// SIMATIC S7-200 project (STEP 7-Micro/WIN), CPU 224XP CN REL 02.01

ORGANIZATION_BLOCK MAIN:OB1
TITLE=PROGRAM COMMENTS
BEGIN
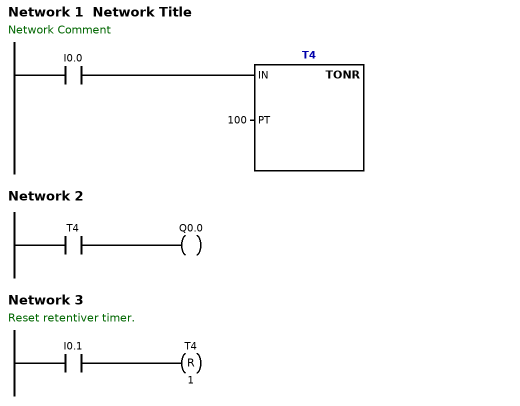
Network 1 // Network Title
// Network Comment
LD     I0.0
TONR   T4, 100
Network 2
LD     T4
=      Q0.0
Network 3
// Reset retentiver timer.
LD     I0.1
R      T4, 1
END_ORGANIZATION_BLOCK
